{attribute 'qualified_only'}
////{xxxattribute 'strict'}
TYPE E_RS_COMM_STATUS :
(
	NOT_INIT	:= -1,
	IDLE		:= 0,
	BUSY		:= 1,
	ERROR		:= 2
);
END_TYPE

(* stored: Version 1.1.0.1, ProductVersion 3.1.4022.16
   DUT E_RS_COMM_STATUS: Id {90ec8231-cc94-48b4-ab64-61ae8346a9fd} *)
